(* IEC 61131-3 sources: eCockpitGit/test_project/src/%F%00 Library/%F%Common Functions/%F%Buffer/%POU%FB_FIFOArray/%PRO%isFull, 1 file *)

(* ---- %GETSET%Get.st ---- *)
//Retruns wether the buffer is full
// |**Version**|**Author**| **Date** |**Changes**
// | 1         | NSN      | 15-02-22 | Creation
VAR
END_VAR

(*%!%__DELIMITER__%!%*)
isFull		:=		S_amount >= S_bufferSize;
